Omron CX-Programmer project NewProject (CX-Programmer 9.81)

# PLC NewPLC1: CJ2M CPU11

## Program NewProgram1 (cyclic task 0)
Local symbols
A1_R1 1.00 BOOL  ; A1 do Relé
B_E 0.00 BOOL  ; Botão Emergência
B_S 0.01 BOOL  ; Botão Stop
B_ST 0.02 BOOL  ; Botão Start
NO_R1 0.03 BOOL  ; NO do Relé

### Section Section1

### Section OUTPUTS

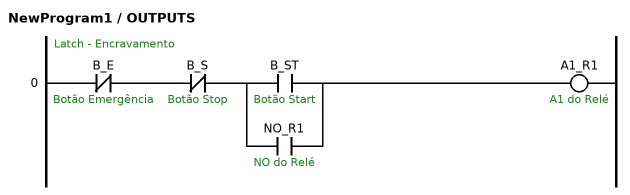
; rung 0: Latch - Encravamento
LDNOT B_E  ; Botão Emergência
ANDNOT B_S  ; Botão Stop
LD B_ST  ; Botão Start
OR NO_R1  ; NO do Relé
ANDLD
OUT A1_R1  ; A1 do Relé

### Section END
; rung 0
END(001)